PROGRAM MAIN
VAR
END_VAR

END_PROGRAM

(* stored: Version 1.1.0.1
   POU MAIN: Id {3b048a0f-5a2a-4132-8784-8a4b2342a2a0} *)
